{attribute 'OPC.UA.DA.StructuredType' := '1'}
FUNCTION_BLOCK FB_GasMonitoringPanel_CDA4022_R2 EXTENDS FB_BaseDevice 

VAR_IN_OUT
	{attribute 'OPC.UA.DA' := '0'}
	fbModbusManager: FB_ModbusManager;
END_VAR

VAR
	// CDA Panel 4022 V3.0 Variables (https://drive.google.com/file/d/1dn1Ot7nd1VML-1RxFooYWTdx5gniYgca/view?usp=sharing)
	(*
	       CO2
		   References - https://iceblast.com.au/wp-content/uploads/2021/03/ABCB-Handbook-Indoor-Air-Quality-2018.pdf   
	*)
	nConcentration_CO2: 	UINT; // reading is value x 10, units are configurable - set to ppm
	nThreshold_CO2_Level1: 	DINT := 800; //ppm (Upper limit of AS 1668.2 recommendation (for CO2 controlled ventilation))
	nAlarm_CO2_Level1: 		UINT; 
	nThreshold_CO2_Level2: 	DINT := 1000; //ppm (ASHRAE 62.1 recommendation (occupant comfort))
	nAlarm_CO2_Level2: 		UINT; 
	nThreshold_CO2_Level3: 	DINT := 5000; //ppm (Australian occupational exposure limit (SWA 2011b) )
	nAlarm_CO2_Level3: 		UINT; 
	
	(*
	       O2
		   References - https://www.cacgas.com.au/blog/bid/378107/oxygen-o2-occupational-health-exposure-standards 
	*)
	nConcentration_O2: 		UINT; // reading is value x 10, units are configurable - set to ppm
	nThreshold_O2_Level1: 	DINT := 195000; //ppm (Minimum "Safe Level")
	nAlarm_O2_Level1: 		UINT; 
	nThreshold_O2_Level2: 	DINT := 160000; //ppm (First signs of anoxia (dizziness, light-headedness))
	nAlarm_O2_Level2: 		UINT; 
	nThreshold_O2_Level3: 	DINT := 235000; //ppm (oxygen levels that exceed 23.5% present a serious fire danger.  At levels of 25%+ items such as clothing can spontaneously combust.  )
	nAlarm_O2_Level3: 		UINT; 	

	// Modbus Variables
	nModbusUnitID: UINT; 
	bFirtRun: BOOL := TRUE;
	bResetTimer: BOOL := TRUE;
	
	// Async Statemachine Variables
	{attribute 'OPC.UA.DA' := '0'}
	eSMState: (WAIT, READ_TRIG, READ, WRITE_TRIG, WRITE, ERROR);
	{attribute 'OPC.UA.DA' := '0'} 
	
	fbTON_DataRefresh: TON := (PT := T#15S, IN := FALSE);
	
	stModRequest_Read_CO2_Actual: ST_Modbus_ReadRequest;
	stModRequest_Read_CO2_AL1: ST_Modbus_ReadRequest;
	stModRequest_Read_CO2_AL2: ST_Modbus_ReadRequest;
	stModRequest_Read_CO2_AL3: ST_Modbus_ReadRequest;
	
	stModRequest_Read_O2_Actual: ST_Modbus_ReadRequest;
	stModRequest_Read_O2_AL1: ST_Modbus_ReadRequest;
	stModRequest_Read_O2_AL2: ST_Modbus_ReadRequest;
	stModRequest_Read_O2_AL3: ST_Modbus_ReadRequest;
	
	
	eOpType: (READ_OP, WRITE_OP);
	{attribute 'OPC.UA.DA' := '0'} 
	bRequestFinished: POINTER TO BOOL;
	{attribute 'OPC.UA.DA' := '0'} 
	bRequestSentToMaster: BOOL 	:= FALSE;
	{attribute 'OPC.UA.DA' := '0'} 
	bRequestCompleted: BOOL 	:= FALSE;
	

	
END_VAR

fbTON_DataRefresh();

IF GVL.bAutoUpdateDeviceState THEN
	eState := eStateTarget;	
END_IF

IF bFirtRun THEN
	init_ModbusRequests();
	bFirtRun := FALSE;
END_IF

IF bResetTimer THEN
	fbTON_DataRefresh.IN := TRUE;
	bResetTimer := FALSE;
END_IF


IF fbTON_DataRefresh.Q THEN
	fbModbusManager.addRequest_Read(ReadRequest := ADR(stModRequest_Read_CO2_Actual));
	fbModbusManager.addRequest_Read(ReadRequest := ADR(stModRequest_Read_CO2_AL1));
	fbModbusManager.addRequest_Read(ReadRequest := ADR(stModRequest_Read_CO2_AL2));
	fbModbusManager.addRequest_Read(ReadRequest := ADR(stModRequest_Read_CO2_AL3));
	fbModbusManager.addRequest_Read(ReadRequest := ADR(stModRequest_Read_O2_Actual));
	fbModbusManager.addRequest_Read(ReadRequest := ADR(stModRequest_Read_O2_AL1));
	fbModbusManager.addRequest_Read(ReadRequest := ADR(stModRequest_Read_O2_AL2));
	fbModbusManager.addRequest_Read(ReadRequest := ADR(stModRequest_Read_O2_AL3));
	
	fbTON_DataRefresh.IN := FALSE;
	bResetTimer := TRUE;
END_IF

nConcentration_CO2 := WORD_TO_UINT(stModRequest_Read_CO2_Actual.ReadRegsVals[1]);
nAlarm_CO2_Level1 := WORD_TO_UINT(stModRequest_Read_CO2_AL1.ReadRegsVals[1]);
nAlarm_CO2_Level2 := WORD_TO_UINT(stModRequest_Read_CO2_AL2.ReadRegsVals[1]);
nAlarm_CO2_Level3 := WORD_TO_UINT(stModRequest_Read_CO2_AL3.ReadRegsVals[1]);

nConcentration_O2 := WORD_TO_UINT(stModRequest_Read_O2_Actual.ReadRegsVals[1]);
nAlarm_O2_Level1 := WORD_TO_UINT(stModRequest_Read_O2_AL1.ReadRegsVals[1]);
nAlarm_O2_Level2 := WORD_TO_UINT(stModRequest_Read_O2_AL2.ReadRegsVals[1]);
nAlarm_O2_Level3 := WORD_TO_UINT(stModRequest_Read_O2_AL3.ReadRegsVals[1]);

METHOD FB_init : BOOL
VAR_INPUT
	bInitRetains : BOOL; // if TRUE, the retain variables are initialized (warm start / cold start)
	bInCopyCode : BOOL;  // if TRUE, the instance afterwards gets moved into the copy code (online change)
	
	ModbusID: UINT;
END_VAR
nModbusUnitID := ModbusID;
END_METHOD

METHOD init_ModbusRequests : BOOL
VAR_INPUT
END_VAR
stModRequest_Read_CO2_Actual.SlaveAddress := nModbusUnitID;			
stModRequest_Read_CO2_Actual.AdrFirstSlaveRegisterRead := 1;
stModRequest_Read_CO2_Actual.QtyWordsToRead := 1;				// The value is a 16-bit word
stModRequest_Read_CO2_Actual.bRequestAccepted := FALSE;
stModRequest_Read_CO2_Actual.bRequestCompleted := FALSE;
stModRequest_Read_CO2_Actual.ReadRegsVals := GVL.ModbusEmptyBuffer;

stModRequest_Read_CO2_AL1.SlaveAddress := nModbusUnitID;			
stModRequest_Read_CO2_AL1.AdrFirstSlaveRegisterRead := 101;
stModRequest_Read_CO2_AL1.QtyWordsToRead := 1;				// The value is a 32-bit word
stModRequest_Read_CO2_AL1.bRequestAccepted := FALSE;
stModRequest_Read_CO2_AL1.bRequestCompleted := FALSE;
stModRequest_Read_CO2_AL1.ReadRegsVals := GVL.ModbusEmptyBuffer;

stModRequest_Read_CO2_AL2.SlaveAddress := nModbusUnitID;			
stModRequest_Read_CO2_AL2.AdrFirstSlaveRegisterRead := 201;
stModRequest_Read_CO2_AL2.QtyWordsToRead := 1;				// The value is a 32-bit word
stModRequest_Read_CO2_AL2.bRequestAccepted := FALSE;
stModRequest_Read_CO2_AL2.bRequestCompleted := FALSE;
stModRequest_Read_CO2_AL2.ReadRegsVals := GVL.ModbusEmptyBuffer;

stModRequest_Read_CO2_AL3.SlaveAddress := nModbusUnitID;			
stModRequest_Read_CO2_AL3.AdrFirstSlaveRegisterRead := 301;
stModRequest_Read_CO2_AL3.QtyWordsToRead := 1;				// The value is a 32-bit word
stModRequest_Read_CO2_AL3.bRequestAccepted := FALSE;
stModRequest_Read_CO2_AL3.bRequestCompleted := FALSE;
stModRequest_Read_CO2_AL3.ReadRegsVals := GVL.ModbusEmptyBuffer;

stModRequest_Read_O2_Actual.SlaveAddress := nModbusUnitID;			
stModRequest_Read_O2_Actual.AdrFirstSlaveRegisterRead := 0;
stModRequest_Read_O2_Actual.QtyWordsToRead := 1;				// The value is a 16-bit word
stModRequest_Read_O2_Actual.bRequestAccepted := FALSE;
stModRequest_Read_O2_Actual.bRequestCompleted := FALSE;
stModRequest_Read_O2_Actual.ReadRegsVals := GVL.ModbusEmptyBuffer;

stModRequest_Read_O2_AL1.SlaveAddress := nModbusUnitID;			
stModRequest_Read_O2_AL1.AdrFirstSlaveRegisterRead := 100;
stModRequest_Read_O2_AL1.QtyWordsToRead := 1;				// The value is a 32-bit word
stModRequest_Read_O2_AL1.bRequestAccepted := FALSE;
stModRequest_Read_O2_AL1.bRequestCompleted := FALSE;
stModRequest_Read_O2_AL1.ReadRegsVals := GVL.ModbusEmptyBuffer;

stModRequest_Read_O2_AL1.SlaveAddress := nModbusUnitID;			
stModRequest_Read_O2_AL1.AdrFirstSlaveRegisterRead := 200;
stModRequest_Read_O2_AL1.QtyWordsToRead := 1;				// The value is a 32-bit word
stModRequest_Read_O2_AL1.bRequestAccepted := FALSE;
stModRequest_Read_O2_AL1.bRequestCompleted := FALSE;
stModRequest_Read_O2_AL1.ReadRegsVals := GVL.ModbusEmptyBuffer;

stModRequest_Read_O2_AL3.SlaveAddress := nModbusUnitID;			
stModRequest_Read_O2_AL3.AdrFirstSlaveRegisterRead := 300;
stModRequest_Read_O2_AL3.QtyWordsToRead := 1;				// The value is a 32-bit word
stModRequest_Read_O2_AL3.bRequestAccepted := FALSE;
stModRequest_Read_O2_AL3.bRequestCompleted := FALSE;
stModRequest_Read_O2_AL3.ReadRegsVals := GVL.ModbusEmptyBuffer;
END_METHOD

END_FUNCTION_BLOCK

(* stored: Version 1.1.0.1, ProductVersion 3.1.4024.12
   POU FB_GasMonitoringPanel_CDA4022_R2: Id {1847ed02-16fe-4e0a-b2f0-be7d20bc131b}, SpecialFunc None
   Method FB_init: Id {bf7737e0-d3a7-46fc-b19f-bb2d92341c1c}
   Method init_ModbusRequests: Id {996ac414-4593-4260-a069-fbb7ff5a9acf} *)
